FUNCTION_BLOCK StorageControl (* Basic FB with empty ECC *)
  (* Standard: 61499-2 *)
  (* Version 1.0, 2021-09-15, dorofeev *)
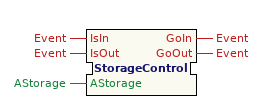
  EVENT_INPUT
    IsIn;
    IsOut;
  END_EVENT
  EVENT_OUTPUT
    GoIn;
    GoOut;
  END_EVENT
  SOCKETS
    AStorage : AStorage;
  END_SOCKETS
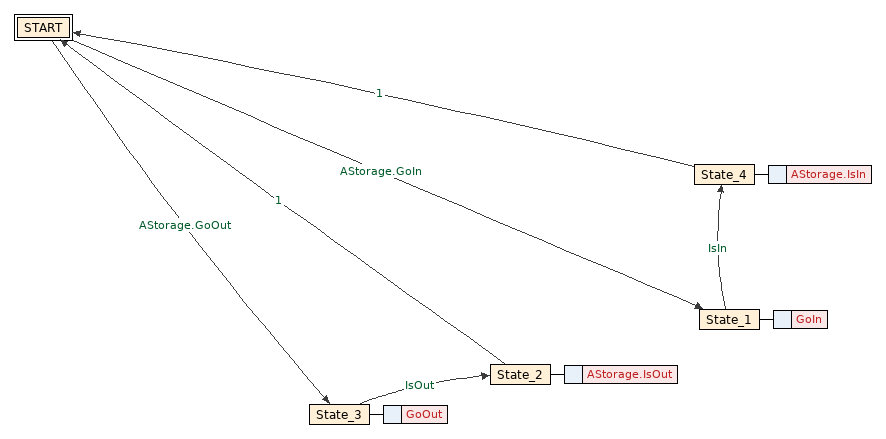
  EC_STATES
    START; (* Initial State *)
    State_1 : -> GoIn;
    State_3 : -> GoOut;
    State_2 : -> AStorage.IsOut;
    State_4 : -> AStorage.IsIn;
  END_STATES
  EC_TRANSITIONS
    State_1 TO State_4 := IsIn;
    State_3 TO State_2 := IsOut;
    START TO State_3 := AStorage.GoOut;
    State_2 TO START := 1;
    START TO State_1 := AStorage.GoIn;
    State_4 TO START := 1;
  END_TRANSITIONS
END_FUNCTION_BLOCK
